Universal Robots URScript: 00B_06_JieXian_ToZero.script

def P00B_06_JieXian_ToZero():
  set_standard_analog_input_domain(0, 1)
  set_standard_analog_input_domain(1, 1)
  set_tool_analog_input_domain(0, 1)
  set_tool_analog_input_domain(1, 1)
  set_analog_outputdomain(0, 0)
  set_analog_outputdomain(1, 0)
  set_tool_voltage(0)
  set_input_actions_to_default()
  set_tcp(p[-0.06448999999999999,0.0207,0.28314999999999996,0.0,0.0,1.5902])
  set_payload(8.0)
  set_safety_mode_transition_hardness(1)
  set_gravity([0.0, 0.0, 9.82])
  $ 1 "机器人程序"
  $ 2 "MoveJ"
  $ 3 "路点_1"
  set_tcp(p[-0.06448999999999999,0.0207,0.28314999999999996,0.0,0.0,1.5902])
  movej(get_inverse_kin(p[.434331656553, .698467371053, .586750973673, -.148550996126, -.158265831010, -1.507060583724], qnear=[1.2589926719665527, -2.003558937703268, -2.0371201674090784, -0.8544166723834437, -1.6501677672015589, 0.3424997925758362]), a=0.6981317007977318, v=0.5235987755982988)
  $ 4 "路点_2"
  set_tcp(p[-0.06448999999999999,0.0207,0.28314999999999996,0.0,0.0,1.5902])
  movej(get_inverse_kin(p[.126979162544, .084230294974, .682340514511, .052958608482, -.000619488234, .974088221183], qnear=[1.6279940605163574, 0.054912447929382324, -2.8315115610705774, -1.888059441243307, -1.5481937567340296, 2.466928005218506]), a=0.6981317007977318, v=0.5235987755982988)
end
